FUNCTION_BLOCK COLOR_GENERATOR
  {SET_ATTRIBUTE(OpcUa, DEVICE.SENSOR)}
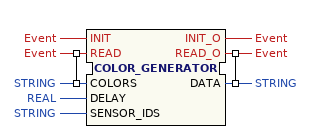
  EVENT_INPUT
    INIT;
    READ WITH COLORS;
  END_EVENT
  EVENT_OUTPUT
    INIT_O;
    READ_O WITH DATA;
  END_EVENT
  VAR_INPUT
    COLORS : STRING;
    DELAY : REAL;
    SENSOR_IDS : STRING;
  END_VAR
  VAR_OUTPUT
    DATA : STRING;
  END_VAR
END_FUNCTION_BLOCK
